{attribute 'GeneratedUsingTerminal: EL6021--0000'}
{attribute addProperty BoxType "EL6021--0000"}
{attribute addProperty Id "EtcSlaveTerminalBaseInputsAT %I*Inputs_6C2FC20224OutputsAT %Q*Outputs_5D00B5E724WcStateAT %I*WcState_9091E0EB2InfoDataAT %I*InfoData_32EB74EA10"}
{attribute addProperty CRC "3795277333"}
{attribute addProperty Size "60"}
TYPE EL6021_E2375615 EXTENDS EtcSlaveTerminalBase :
STRUCT
	{attribute addProperty Name "Inputs"}
	Inputs : Inputs_6C2FC202;
	{attribute addProperty Name "Outputs"}
	Outputs : Outputs_5D00B5E7;
	{attribute addProperty Name "WcState"}
	WcState : WcState_9091E0EB;
	{attribute addProperty Name "InfoData"}
	InfoData : InfoData_32EB74EA;
END_STRUCT
END_TYPE

(* stored: Version 1.2.0.0, ProductVersion 3.1.4024.9
   DUT EL6021_E2375615: Id {f07115e7-8cdb-4499-9121-0dfe85a0b7f8} *)
